{attribute 'Tc2GvlVarNames'}
{attribute 'strict'}
//Stato del WorkAreaManager
TYPE e_Stato_WAManager :
(
	WAMANAGER_NOT_DEFINED						:= -1,
	(*********************************************************************)
	WAMANAGER_NOP								:= 100,
	(*********************************************************************)
	WAMANAGER_CICLO_RIPOSO_INIT					:= 110,
	WAMANAGER_CICLO_RIPOSO_RUN					:= 111,
	WAMANAGER_CICLO_RIPOSO_END					:= 112,
	(*********************************************************************)
	//WAMANAGER_CICLO_PALL_INIT					:= 120,
	//WAMANAGER_CICLO_PRELIEVO_PALL_RUN			:= 121,
	//WAMANAGER_CICLO_PRELIEVO_PALL_END			:= 122,
	//WAMANAGER_CICLO_DEPOSITO_PALL_RUN			:= 123,
	//WAMANAGER_CICLO_DEPOSITO_PALL_END			:= 124,
	(*********************************************************************)
	//WAMANAGER_CICLO_FALDA_VUOTI_INIT			:= 130,
	//WAMANAGER_CICLO_PRELIEVO_FALDA_VUOTI_RUN	:= 131,
	//WAMANAGER_CICLO_PRELIEVO_FALDA_VUOTI_END	:= 132,
	//WAMANAGER_CICLO_DEPOSITO_FALDA_VUOTI_RUN	:= 133,
	//WAMANAGER_CICLO_DEPOSITO_FALDA_VUOTI_END	:= 134,
	(*********************************************************************)
	WAMANAGER_CICLO_FALDA_INIT					:= 140,
	WAMANAGER_CICLO_PRELIEVO_FALDA_RUN			:= 141,
	WAMANAGER_CICLO_PRELIEVO_FALDA_END			:= 142,
	WAMANAGER_CICLO_DEPOSITO_FALDA_RUN			:= 143,
	WAMANAGER_CICLO_DEPOSITO_FALDA_END			:= 144,
	(*********************************************************************)
	//WAMANAGER_CICLO_PACCO_INIT					:= 150,
	//WAMANAGER_CICLO_PRELIEVO_PACCO_RUN			:= 151,
	//WAMANAGER_CICLO_PRELIEVO_PACCO_END			:= 152,
	//WAMANAGER_CICLO_DEPOSITO_PACCO_RUN			:= 153,
	//WAMANAGER_CICLO_DEPOSITO_PACCO_END			:= 154,
	(*********************************************************************)
	(* Ciclo Lastra NORMALE..Prelievo in Pick-Point *)
	WAMANAGER_CICLO_LASTRA_PP_INIT				:= 160, 
	WAMANAGER_CICLO_PRELIEVO_LASTRA_PP_RUN		:= 161,
	WAMANAGER_CICLO_PRELIEVO_LASTRA_PP_END		:= 162,
	WAMANAGER_CICLO_DEPOSITO_LASTRA_PP_RUN		:= 163,
	WAMANAGER_CICLO_DEPOSITO_LASTRA_PP_END		:= 164,
	(*********************************************************************)
	(* Ciclo Lastra SPECIALE..Prelievo in Work-Area *)
	WAMANAGER_CICLO_LASTRA_WA_INIT				:= 170,
	WAMANAGER_CICLO_PRELIEVO_LASTRA_WA_RUN		:= 171,
	WAMANAGER_CICLO_PRELIEVO_LASTRA_WA_END		:= 172,
	WAMANAGER_CICLO_DEPOSITO_LASTRA_WA_RUN		:= 173,
	WAMANAGER_CICLO_DEPOSITO_LASTRA_WA_END		:= 174,
	
	WAMANAGER_CICLO_DEPOSITO_LASTRA_SU_PAREGGIATORE_RUN		:= 180,
	WAMANAGER_CICLO_DEPOSITO_LASTRA_SU_PAREGGIATORE_END		:= 181,
	
	WAMANAGER_CICLO_PAREGGIATURA_RUN		:= 182,
	WAMANAGER_CICLO_PAREGGIATURA_END		:= 183,
	
	WAMANAGER_CICLO_PRELIEVO_LASTRA_DA_PAREGGIATORE_RUN		:= 184,
	WAMANAGER_CICLO_PRELIEVO_LASTRA_DA_PAREGGIATORE_END		:= 185,
	
	(* Ciclo lastra per depalettizzare da postazioni senza formature, con autoapprndimenti*)
	WAMANAGER_CICLO_LASTRA_DEPAL_INIT  			:= 190,
	WAMANAGER_CICLO_PRELIEVO_LASTRA_DEPAL_RUN	:= 191,
	WAMANAGER_CICLO_PRELIEVO_LASTRA_DEPAL_END	:= 192,
	(* Ciclo lastra deposito su rulliera *)
	WAMANAGER_CICLO_DEPOSITO_LASTRA_DEPAL_RUN	:= 193,
	WAMANAGER_CICLO_DEPOSITO_LASTRA_DEPAL_END	:= 194,
	(* Ciclo deposito FALDA su magazzino dedicato *)
	WAMANAGER_CICLO_DEPOSITO_FALDA_DEPAL_RUN 	:= 195,
	WAMANAGER_CICLO_DEPOSITO_FALDA_DEPAL_END    := 196,
	
	(*********************************************************************)	
	WAMANAGER_SALTA_DA_RIPOSO_A_PRELIEVO		:= 200
);
END_TYPE
//  WAMANAGER_NOT_DEFINED = '-1'

(* stored: Version 1.1.0.1, ProductVersion 3.1.4024.11
   EnumerationTextList e_Stato_WAManager: Id {dafd2037-31e3-4743-8613-215615a35dd7} *)
